KUKA KRL program: DEXTERITYTEST.src, DEXTERITYTEST.dat

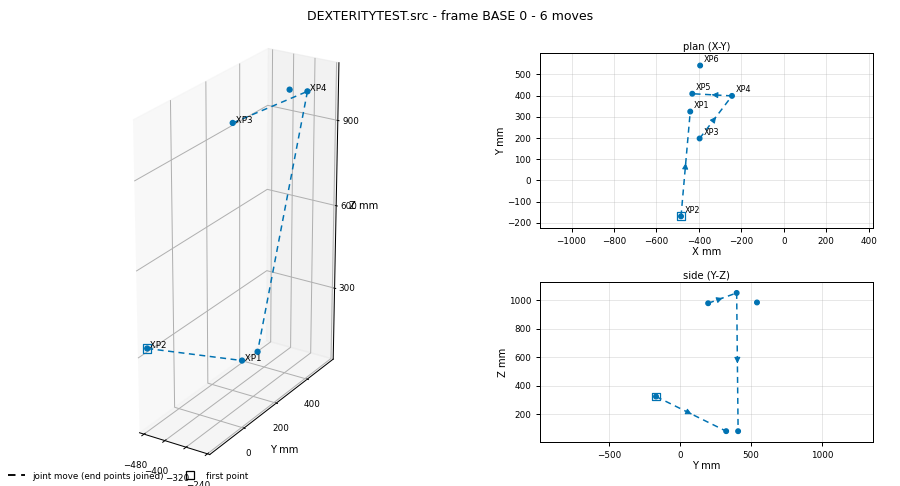
[picture p0: tool path of DEXTERITYTEST.src in frame BASE 0, 6 of 8 moves have a stored position in this frame; points joined in program order, loops and branches not executed]
--- DEXTERITYTEST.src ---
&ACCESS RVP
&REL 286
&PARAM TEMPLATE = C:\KRC\Roboter\Template\vorgabe
&PARAM EDITMASK = *
DEF DEXTERITYTEST( )
DECL BOOL TEMP, HEMP, SEMP, REMP
INT X, n, result
DECL INT md_int[16]
DECL REAL md_real[16]
;FOLD INI
  ;FOLD BASISTECH INI
    GLOBAL INTERRUPT DECL 3 WHEN $STOPMESS==TRUE DO IR_STOPM ( )
    INTERRUPT ON 3
    BAS (#INITMOV,0 )
  ;ENDFOLD (BASISTECH INI)
  ;FOLD USER INI
    ;Make your modifications here

  ;ENDFOLD (USER INI)
   LOGROBOTDATA=TRUE
   SERVERCONNECTED=TRUE
   TCPCONNECTION=FALSE
;ENDFOLD (INI)

$TOOL=TOOL_DATA[5]
$VEL.CP=1.0
$VEL.ORI1=100
$VEL.ORI2=100
$ACC.CP=1.0
$ACC.ORI1=80
$ACC.ORI2=80
FOR X=1 TO 6
$ACC_AXIS[X]=70
$VEL_AXIS[X]=70
ENDFOR

CANDLE()

$OV_PRO=8

;FOLD PTP P2 Vel=100 % PDAT2 Tool[5]:Pneumatic_gripper_probe Base[0];%{PE}%R 5.6.11,%MKUKATPBASIS,%CMOVE,%VPTP,%P 1:PTP, 2:P2, 3:, 5:100, 7:PDAT2
$BWDSTART=FALSE
PDAT_ACT=PPDAT2
FDAT_ACT=FP2
BAS(#PTP_PARAMS,100)
PTP XP2
;ENDFOLD

;FOLD PTP P1 Vel=100 % PDAT1 Tool[5]:Pneumatic_gripper_probe Base[0];%{PE}%R 5.6.11,%MKUKATPBASIS,%CMOVE,%VPTP,%P 1:PTP, 2:P1, 3:, 5:100, 7:PDAT1
$BWDSTART=FALSE
PDAT_ACT=PPDAT1
FDAT_ACT=FP1
BAS(#PTP_PARAMS,100)
PTP XP1
;ENDFOLD

;FORCE ON RED DOTS
;FOR X=1 TO 8
  ;TEMP=TRIG()
  ;TEMP=SETSTIFF("Z", 10.0)
  ;TEMP=SETFORCE("Z", 68.85)
  ;LIN_REL{Y 1}
  ;LIN_REL{Z 100}
  ;WAIT SEC 2
  ;LIN_REL{Y -1}
  ;TEMP=FORCEZSTOP()
  ;PTP $POS_ACT_MES
  ;$STIFFNESS.STRATEGY=10
  ;$STIFFNESS.COMMIT=TRUE
;ENDFOR

;FOR CONSTANT FORCE
TEMP=TRIG()
HEMP=SETSTIFF("Z", 10.0)
SEMP=SETFORCE("Z", 68.65)

LIN_REL{Y 1}
LIN_REL{Z 800}

REMP=FORCEZSTOP()

FOR n=1 TO 16
  md_int[n]=0
  md_real[n]=0
ENDFOR

md_real[1]=0.01

result=MD_CMD("PAPAS","TRIGBYCONTACT",md_int[],md_real[])

PTP $POS_ACT_MES

$STIFFNESS.STRATEGY=10
$STIFFNESS.COMMIT=TRUE

;FOLD PTP P3 Vel=100 % PDAT3 Tool[5]:Pneumatic_gripper_probe Base[0];%{PE}%R 5.6.11,%MKUKATPBASIS,%CMOVE,%VPTP,%P 1:PTP, 2:P3, 3:, 5:100, 7:PDAT3
$BWDSTART=FALSE
PDAT_ACT=PPDAT3
FDAT_ACT=FP3
BAS(#PTP_PARAMS,100)
PTP XP3
;ENDFOLD

CANDLE()

;FOLD PTP P4 Vel=100 % PDAT12 Tool[5]:Pneumatic_gripper_probe Base[0];%{PE}%R 5.6.11,%MKUKATPBASIS,%CMOVE,%VPTP,%P 1:PTP, 2:P4, 3:, 5:100, 7:PDAT12
$BWDSTART=FALSE
PDAT_ACT=PPDAT12
FDAT_ACT=FP4
BAS(#PTP_PARAMS,100)
PTP XP4
;ENDFOLD

;FOLD PTP P5 Vel=100 % PDAT11 Tool[5]:Pneumatic_gripper_probe Base[0];%{PE}%R 5.6.11,%MKUKATPBASIS,%CMOVE,%VPTP,%P 1:PTP, 2:P5, 3:, 5:100, 7:PDAT11
$BWDSTART=FALSE
PDAT_ACT=PPDAT11
FDAT_ACT=FP5
BAS(#PTP_PARAMS,100)
PTP XP5
;ENDFOLD

TEMP=TRIG()
HEMP=SETSTIFF("Y", 10.0)
SEMP=SETFORCE("Y", 68.65)

LIN_REL{Y -2}
LIN_REL{Z 800}

REMP=FORCEZSTOP()

PTP $POS_ACT_MES

$STIFFNESS.STRATEGY=10
$STIFFNESS.COMMIT=TRUE

$OV_PRO=25

;FOLD PTP P6 Vel=100 % PDAT13 Tool[5]:Pneumatic_gripper_probe Base[0];%{PE}%R 5.6.11,%MKUKATPBASIS,%CMOVE,%VPTP,%P 1:PTP, 2:P6, 3:, 5:100, 7:PDAT13
$BWDSTART=FALSE
PDAT_ACT=PPDAT13
FDAT_ACT=FP6
BAS(#PTP_PARAMS,100)
PTP XP6
;ENDFOLD

CANDLE()

LOGROBOTDATA=FALSE
SERVERCONNECTED=FALSE
TCPCONNECTION=FALSE

END

--- DEXTERITYTEST.dat ---
&ACCESS RVP
&REL 286
&PARAM TEMPLATE = C:\KRC\Roboter\Template\vorgabe
&PARAM EDITMASK = *
DEFDAT  DEXTERITYTEST
;FOLD EXTERNAL DECLARATIONS;%{PE}%MKUKATPBASIS,%CEXT,%VCOMMON,%P
;FOLD BASISTECH EXT;%{PE}%MKUKATPBASIS,%CEXT,%VEXT,%P
EXT  BAS (BAS_COMMAND  :IN,REAL  :IN )
DECL INT SUCCESS
;ENDFOLD (BASISTECH EXT)
;FOLD USER EXT;%{E}%MKUKATPUSER,%CEXT,%VEXT,%P
;Make here your modifications

;ENDFOLD (USER EXT)
;ENDFOLD (EXTERNAL DECLARATIONS)
DECL BASIS_SUGG_T LAST_BASIS={POINT1[] "P6                      ",POINT2[] "P6                      ",CP_PARAMS[] "CPDAT0                  ",PTP_PARAMS[] "PDAT13                  ",CONT[] "                        ",CP_VEL[] "2.0                     ",PTP_VEL[] "100                     ",SYNC_PARAMS[] "SYNCDAT                 ",SPL_NAME[] "S0                      "}
DECL E6POS XP1={X -440.843811,Y 324.556305,Z 79.5063934,A 18.0319691,B 89.5150909,C -72.4470367,S 1,T 44,E1 -44.7626114,E2 0.0,E3 0.0,E4 0.0,E5 0.0,E6 0.0}
DECL FDAT FP1={TOOL_NO 5,BASE_NO 0,IPO_FRAME #BASE,POINT2[] " ",TQ_STATE FALSE}
DECL PDAT PPDAT1={VEL 100.0,ACC 100.0,APO_DIST 100.0,APO_MODE #CPTP}
DECL E6POS XP2={X -484.350403,Y -169.003296,Z 323.053589,A 179.172501,B -1.544963,C -179.079605,S 1,T 4,E1 -33.3453293,E2 0.0,E3 0.0,E4 0.0,E5 0.0,E6 0.0}
DECL FDAT FP2={TOOL_NO 5,BASE_NO 0,IPO_FRAME #BASE,POINT2[] " ",TQ_STATE FALSE}
DECL PDAT PPDAT2={VEL 100.0,ACC 100.0,APO_DIST 100.0,APO_MODE #CPTP}
DECL E6POS XP3={X -396.731201,Y 197.784302,Z 979.372986,A 175.080093,B 74.0202026,C 80.7419205,S 1,T 44,E1 -44.761879,E2 0.0,E3 0.0,E4 0.0,E5 0.0,E6 0.0}
DECL FDAT FP3={TOOL_NO 5,BASE_NO 0,IPO_FRAME #BASE,POINT2[] " ",TQ_STATE FALSE}
DECL PDAT PPDAT3={VEL 100.0,ACC 100.0,APO_DIST 100.0,APO_MODE #CPTP}
DECL E6POS XP4={X -244.282394,Y 398.385712,Z 1051.89404,A 71.0968704,B -33.2627602,C -73.0887985,S 2,T 8,E1 -15.1787796,E2 0.0,E3 0.0,E4 0.0,E5 0.0,E6 0.0}
DECL FDAT FP4={TOOL_NO 5,BASE_NO 0,IPO_FRAME #BASE,POINT2[] " ",TQ_STATE FALSE}
DECL PDAT PPDAT4={VEL 100.0,ACC 100.0,APO_DIST 100.0,APO_MODE #CPTP}
DECL E6POS XP5={X -431.315094,Y 408.537811,Z 79.2730637,A 14.4738703,B 86.6407471,C -166.428406,S 2,T 8,E1 2.76114702,E2 0.0,E3 0.0,E4 0.0,E5 0.0,E6 0.0}
DECL FDAT FP5={TOOL_NO 5,BASE_NO 0,IPO_FRAME #BASE,POINT2[] " ",TQ_STATE FALSE}
DECL PDAT PPDAT5={VEL 100.0,ACC 100.0,APO_DIST 100.0,APO_MODE #CPTP}
DECL E6POS XP6={X -394.255707,Y 541.328796,Z 984.919312,A 149.836105,B 74.7782516,C -6.15868378,S 2,T 8,E1 2.836447,E2 0.0,E3 0.0,E4 0.0,E5 0.0,E6 0.0}
DECL FDAT FP6={TOOL_NO 5,BASE_NO 0,IPO_FRAME #BASE,POINT2[] " ",TQ_STATE FALSE}
DECL PDAT PPDAT6={VEL 100.0,ACC 100.0,APO_DIST 100.0,APO_MODE #CPTP}
DECL PDAT PPDAT7={VEL 100.0,ACC 100.0,APO_DIST 100.0,APO_MODE #CPTP}
DECL PDAT PPDAT8={VEL 100.0,ACC 100.0,APO_DIST 100.0,APO_MODE #CPTP}
DECL PDAT PPDAT9={VEL 100.0,ACC 100.0,APO_DIST 100.0,APO_MODE #CPTP}
DECL PDAT PPDAT10={VEL 100.0,ACC 100.0,APO_DIST 100.0,APO_MODE #CPTP}
DECL PDAT PPDAT11={VEL 100.0,ACC 100.0,APO_DIST 100.0,APO_MODE #CPTP}
DECL PDAT PPDAT12={VEL 100.0,ACC 100.0,APO_DIST 100.0,APO_MODE #CPTP}
DECL PDAT PPDAT13={VEL 100.0,ACC 100.0,APO_DIST 100.0,APO_MODE #CPTP}
ENDDAT
